(* Logix 5000 project; controller Comas_L4 vendor 1 type 14 code 193 rev 30.11; software revision 30.02; part 4 of 12 *)

ADD_ON_INSTRUCTION Output_Cams   (* revision 1.1, vendor Rockwell Automation *)
// Help:
// Cet Add-On permet la gestion d'une sortie commandée en fonction de la position d'un axe.
// Entre autre, la gestion des temps de réaction est prise en compte pour  le On/Off de la sortie.( Compensation du temps mort).
// La OutputCam est commandée quelque soit le sens de rotation de l'axe.( Bidirectionnal)
// Les entrées :
// In_ServoPosAxe_02.CommandPosition
VAR_INPUT
   Cmd_Enable_AOI : BOOL; {required}   // Entrée de Validation Du Fonctionnement De Output_Cam
   In_ServoPos : REAL; {required}   // Entrée de la Position de l'axe, préferez la Position Commandée
   In_ServoVel : REAL; {required}   // Entrée de la Vitesse de l'axe, Préferez la vitesse commandée
   Set_Period : REAL; {required}   // Entrée pour la Période de l'axe (Unwind Position) pour un axe rotatif. Pour un Axe Linéaire, Entrez ZERO comme valeur
   Set_OnPos : REAL; {required}   // Entrée pour la position de mise à UN de OuputCam
   Set_OffPos : REAL; {required}   // Entrée pour la position de mise à ZERO de OuputCam
   Set_TCompOn : DINT; {required}   // Entrée pour le temps de réaction de mise à UN des Actionneur/Pré-actionneur. ( en ms)
   Set_TCompOff : DINT; {required}   // Entrée pour le temps de réaction de mise à ZERO des Actionneur/Pré-actionneur.( en ms)
END_VAR
VAR_OUTPUT
   Out_Cam : BOOL; {access Read Only, required}   // Sotrie de la OutputCam
END_VAR
VAR
   L_OffPos : REAL;   // Pour Calcul de la position On avec Compensation du temps Mort
   L_OnPos : REAL;   // Pour Calcul de la position Off avec Compensation du temps Mort
END_VAR

ROUTINE Logic   (* structured text *)
   (*
   
   		Historic :
   
   					02.11.2008	PLM		Creation
   
   		Topic : This Add_On allows to switch On and Off anOutput and this related to the position of an Axis.
   				The deadTime compesation is taken into account ;
   *)
   
   
   
   	IF Cmd_Enable_AOI THEN
   
   		L_OnPos			:= Set_OnPos - (Set_TCompOn*In_ServoVel/1000);
   		IF L_OnPos < 0 THEN
   			L_OnPos			:= L_OnPos+Set_Period;
   		ELSIF L_OnPos > Set_Period THEN
   			L_OnPos			:= L_OnPos-Set_Period;
   		END_IF;
   
   
   		L_OffPos			:= Set_OffPos - (Set_TCompOff*In_ServoVel/1000);
   			IF L_OffPos < 0 THEN
   			L_OffPos		:= L_OffPos+Set_Period;
   		ELSIF L_OffPos > Set_Period THEN
   			L_OffPos		:= L_OffPos-Set_Period;
   		END_IF;
   
   		IF L_OnPos > L_OffPos THEN
   			IF In_ServoPos > L_OnPos OR In_ServoPos < L_OffPos THEN
   				Out_Cam		:= 1;
   			ELSE
   				Out_Cam		:= 0;
   			END_IF ;
   		ELSE
   			IF In_ServoPos > L_OnPos AND In_ServoPos < L_OffPos THEN
   				Out_Cam		:= 1;
   			ELSE
   				Out_Cam		:= 0;
   			END_IF ;
   		END_IF;
   	ELSE
   		Out_Cam				:= 0;
   	END_IF;
END_ROUTINE
END_ADD_ON_INSTRUCTION

ADD_ON_INSTRUCTION Pilotage_Relatif   (* revision 1.5 *)
// Revision note:
// V1.5: Guy : Mouvement incrémental
// V1.4: Guy : Simplification
// V1.3: Ajout:
//  tolérance, axe modulo
// V1.2: Avec mode de positionnement
// V1.1: Correction du double MSO
//    ( double appel de bloc)
// V1.0: Depart
VAR_IN_OUT
   MVT_Axe : AXIS_CIP_DRIVE; {required}   // Axe esclave a controler
END_VAR
VAR_INPUT
   MVT_Activation : BOOL; {required}   // Activation puissance A Activer avant d'engager
   MVT_Val_Position : REAL; {required}   // Position Cible
   MVT_Val_Vitesse : REAL; {required}   // Valeur de vitesse global de l'axe
   MVT_Val_Acc : REAL; {required}   // Valeur d accel gloable de laxe
   MVT_Val_Dec : REAL; {required}   // Valeur de decel
   MVT_Val_Jerk : REAL; {required}   // Valeur de jerk
END_VAR
VAR_OUTPUT
   MVT_ER : BOOL; {access Read Only, visible}   // Erreur dans le module
   MVT_En_Pos : BOOL; {visible}   // En position
END_VAR
VAR_INPUT
   MVT_Mode_Positionnement : DINT; {required}   // Mode de positionnement
   MVT_Tolerance_Arret : REAL; {required}   // tolerance d'arret
   MVT_Axe_Modulo : BOOL; {required}   // = 1 axe modulo
   MVT_Val_Modulo : DINT; {required}   // valeur du modulo
END_VAR
VAR_OUTPUT
   MVT_Axe_En_Mvt : BOOL; {access Read Only, visible}   // Axe en mouvement
END_VAR
VAR_INPUT
   MVT_Start : BOOL; {required}
END_VAR
VAR
   MVT_MSO_activation : MOTION_INSTRUCTION; {access None}
   MVT_Axe_Active : BOOL; {access None}
   MVT_MSO_desactivation : MOTION_INSTRUCTION; {access None}
   MVT_Val_Position_Neg : REAL; {access None}
   MVT_Val_Position_Pos : REAL; {access None}
   MVT_Commande_Mouvement : BOOL; {access None}
   MVT_MAM_Axe : MOTION_INSTRUCTION; {access None}
   MVT_MSO_desactivation2 : MOTION_INSTRUCTION; {access None}
   MVT_Val_Position_Neg_mod : REAL; {access None}
   MVT_Val_Position_Pos_mod : REAL; {access None}
   MVT_En_Pos_sans_modulo : BOOL; {access None}
   MVT_En_Pos_modulo : BOOL; {access None}
   MVT_Front_arret : BOOL; {access None}
   MVT_MAS_Axe : MOTION_INSTRUCTION; {access None}
   Front_Raz_Position : BOOL; {access None}
   MVT_Tempo_Axe_Actif : TIMER; {access None}
   MVT_Tempo_Axe_Actif_MSF : TIMER; {access None}
   Axe_En_Pos : BOOL; {access None}
   Etape_MAM : DINT; {access None}
   Frt_MAM_dn : BOOL; {access None}
   Frt_MAM_IP : BOOL; {access None}
   MVT_MAS : MOTION_INSTRUCTION; {access None}
END_VAR

ROUTINE Logic   (* ladder *)
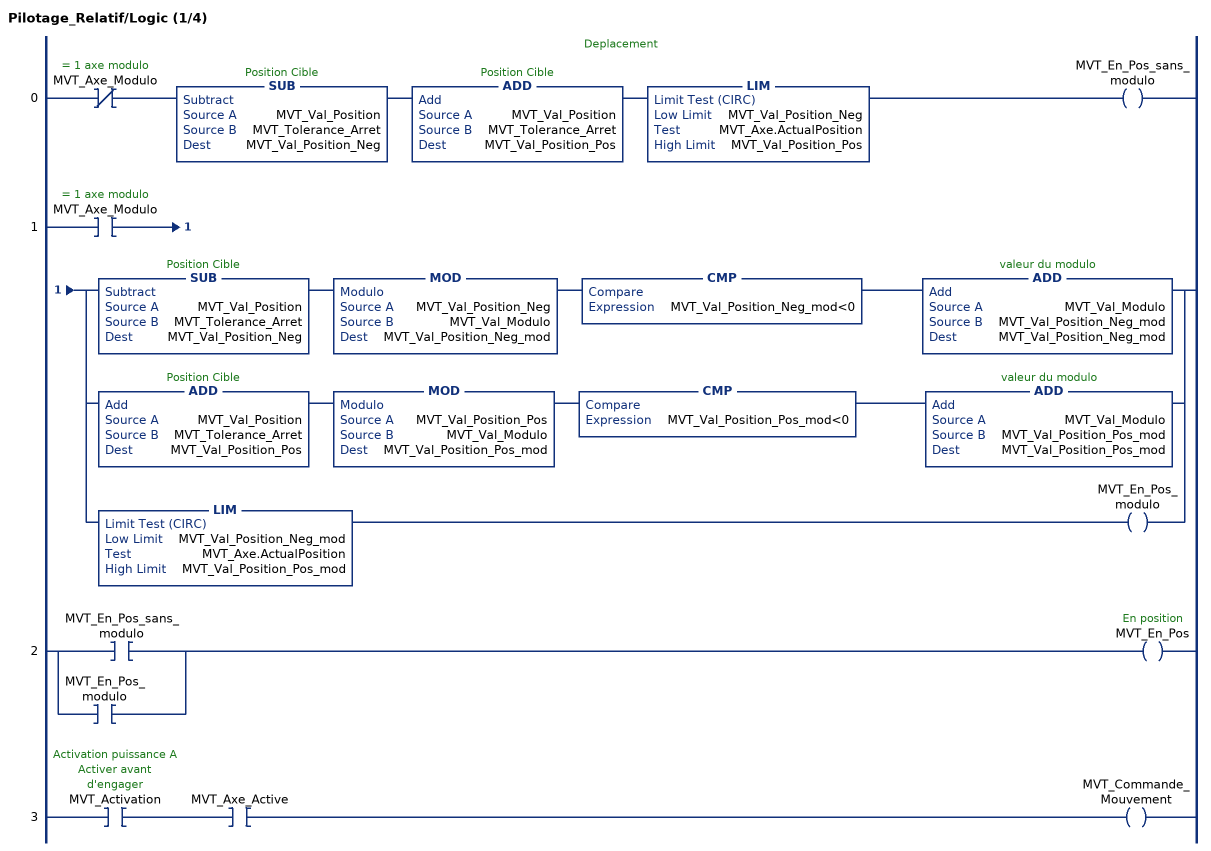
   // Deplacement
   0: XIO(MVT_Axe_Modulo)SUB(MVT_Val_Position,MVT_Tolerance_Arret,MVT_Val_Position_Neg)ADD(MVT_Val_Position,MVT_Tolerance_Arret,MVT_Val_Position_Pos)LIM(MVT_Val_Position_Neg,MVT_Axe.ActualPosition,MVT_Val_Position_Pos)OTE(MVT_En_Pos_sans_modulo);
   1: XIC(MVT_Axe_Modulo)[SUB(MVT_Val_Position,MVT_Tolerance_Arret,MVT_Val_Position_Neg) MOD(MVT_Val_Position_Neg,MVT_Val_Modulo,MVT_Val_Position_Neg_mod) CMP(MVT_Val_Position_Neg_mod<0) ADD(MVT_Val_Modulo,MVT_Val_Position_Neg_mod,MVT_Val_Position_Neg_mod) ,ADD(MVT_Val_Position,MVT_Tolerance_Arret,MVT_Val_Position_Pos) MOD(MVT_Val_Position_Pos,MVT_Val_Modulo,MVT_Val_Position_Pos_mod) CMP(MVT_Val_Position_Pos_mod<0) ADD(MVT_Val_Modulo,MVT_Val_Position_Pos_mod,MVT_Val_Position_Pos_mod) ,LIM(MVT_Val_Position_Neg_mod,MVT_Axe.ActualPosition,MVT_Val_Position_Pos_mod) OTE(MVT_En_Pos_modulo) ];
   2: [XIC(MVT_En_Pos_sans_modulo) ,XIC(MVT_En_Pos_modulo) ]OTE(MVT_En_Pos);
   3: XIC(MVT_Activation)XIC(MVT_Axe_Active)OTE(MVT_Commande_Mouvement);
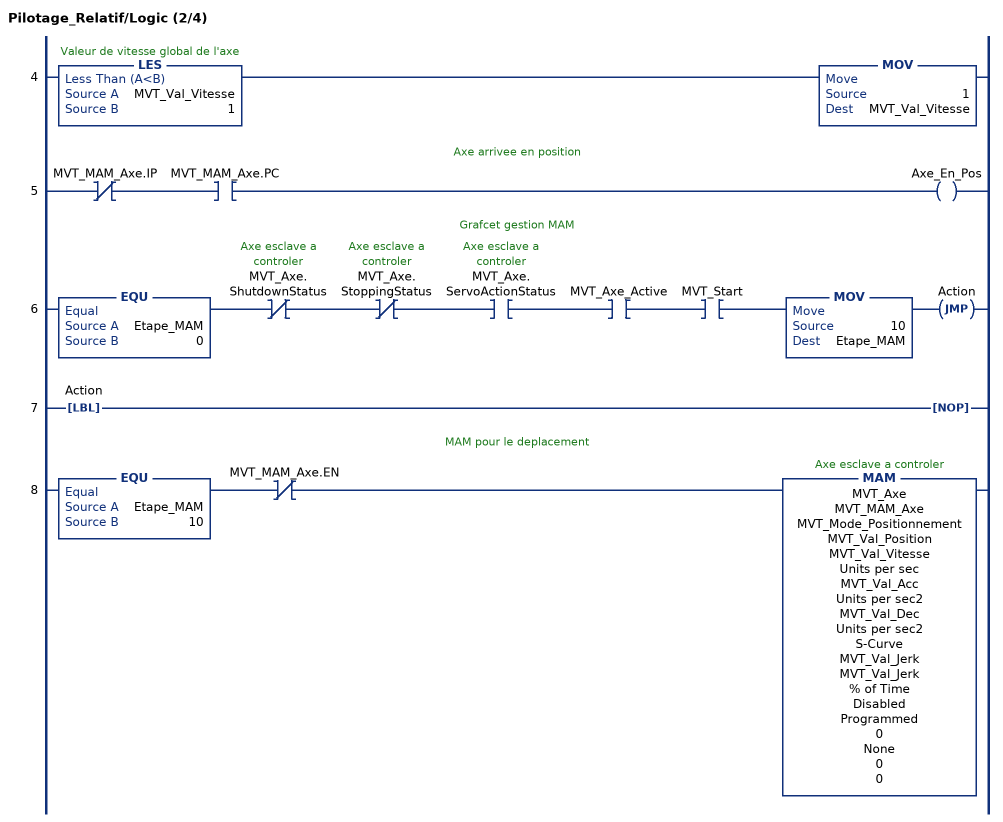
   4: LES(MVT_Val_Vitesse,1)MOV(1,MVT_Val_Vitesse);
   // Axe arrivee en position
   5: XIO(MVT_MAM_Axe.IP)XIC(MVT_MAM_Axe.PC)OTE(Axe_En_Pos);
   // Grafcet gestion MAM
   6: EQU(Etape_MAM,0)XIO(MVT_Axe.ShutdownStatus)XIO(MVT_Axe.StoppingStatus)XIC(MVT_Axe.ServoActionStatus)XIC(MVT_Axe_Active)XIC(MVT_Start)MOV(10,Etape_MAM)JMP(Action);
   7: LBL(Action)NOP();
   // MAM pour le deplacement
   8: EQU(Etape_MAM,10)XIO(MVT_MAM_Axe.EN)MAM(MVT_Axe,MVT_MAM_Axe,MVT_Mode_Positionnement,MVT_Val_Position,MVT_Val_Vitesse,Units per sec,MVT_Val_Acc,Units per sec2,MVT_Val_Dec,Units per sec2,S-Curve,MVT_Val_Jerk,MVT_Val_Jerk,% of Time,Disabled,Programmed,0,None,0,0);
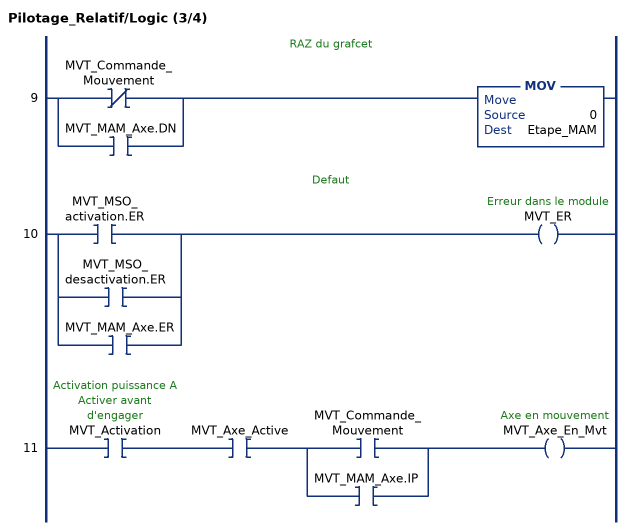
   // RAZ du grafcet
   9: [XIO(MVT_Commande_Mouvement) ,XIC(MVT_MAM_Axe.DN) ]MOV(0,Etape_MAM);
   // Defaut
   10: [XIC(MVT_MSO_activation.ER) ,XIC(MVT_MSO_desactivation.ER) ,XIC(MVT_MAM_Axe.ER) ]OTE(MVT_ER);
   11: XIC(MVT_Activation)XIC(MVT_Axe_Active)[XIC(MVT_Commande_Mouvement) ,XIC(MVT_MAM_Axe.IP) ]OTE(MVT_Axe_En_Mvt);
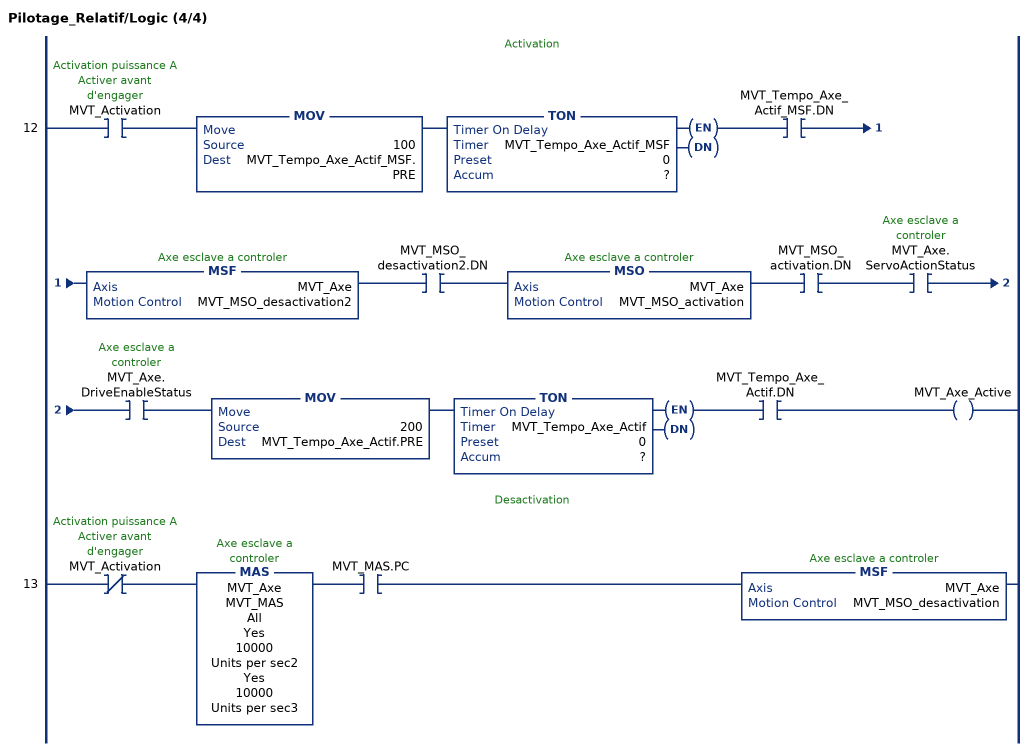
   // Activation
   12: XIC(MVT_Activation)MOV(100,MVT_Tempo_Axe_Actif_MSF.PRE)TON(MVT_Tempo_Axe_Actif_MSF,?,?)XIC(MVT_Tempo_Axe_Actif_MSF.DN)MSF(MVT_Axe,MVT_MSO_desactivation2)XIC(MVT_MSO_desactivation2.DN)MSO(MVT_Axe,MVT_MSO_activation)XIC(MVT_MSO_activation.DN)XIC(MVT_Axe.ServoActionStatus)XIC(MVT_Axe.DriveEnableStatus)MOV(200,MVT_Tempo_Axe_Actif.PRE)TON(MVT_Tempo_Axe_Actif,?,?)XIC(MVT_Tempo_Axe_Actif.DN)OTE(MVT_Axe_Active);
   // Desactivation
   13: XIO(MVT_Activation)MAS(MVT_Axe,MVT_MAS,All,Yes,10000,Units per sec2,Yes,10000,Units per sec3)XIC(MVT_MAS.PC)MSF(MVT_Axe,MVT_MSO_desactivation);
END_ROUTINE
END_ADD_ON_INSTRUCTION

ADD_ON_INSTRUCTION Pilotage_Relatif_Virtuel   (* revision 1.5 *)
// Revision note:
// V1.5: Guy : Mouvement incrémental
// V1.4: Guy : Simplification
// V1.3: Ajout:
//  tolérance, axe modulo
// V1.2: Avec mode de positionnement
// V1.1: Correction du double MSO
//    ( double appel de bloc)
// V1.0: Depart
VAR_IN_OUT
   MVT_Axe : AXIS_VIRTUAL; {required}   // Axe esclave a controler
END_VAR
VAR_INPUT
   MVT_Activation : BOOL; {required}   // Activation puissance A Activer avant d'engager
   MVT_Val_Position : REAL; {required}   // Position Cible
   MVT_Val_Vitesse : REAL; {required}   // Valeur de vitesse global de l'axe
   MVT_Val_Acc : REAL; {required}   // Valeur d accel gloable de laxe
   MVT_Val_Dec : REAL; {required}   // Valeur de decel
   MVT_Val_Jerk : REAL; {required}   // Valeur de jerk
END_VAR
VAR_OUTPUT
   MVT_ER : BOOL; {access Read Only, visible}   // Erreur dans le module
   MVT_En_Pos : BOOL; {visible}   // En position
END_VAR
VAR_INPUT
   MVT_Mode_Positionnement : DINT; {required}   // Mode de positionnement
   MVT_Tolerance_Arret : REAL; {required}   // tolerance d'arret
   MVT_Axe_Modulo : BOOL; {required}   // = 1 axe modulo
   MVT_Val_Modulo : DINT; {required}   // valeur du modulo
END_VAR
VAR_OUTPUT
   MVT_Axe_En_Mvt : BOOL; {access Read Only, visible}   // Axe en mouvement
END_VAR
VAR_INPUT
   MVT_Start : BOOL; {required}
END_VAR
VAR
   MVT_Axe_Active : BOOL; {access None}
   MVT_Val_Position_Neg : REAL; {access None}
   MVT_Val_Position_Pos : REAL; {access None}
   MVT_Commande_Mouvement : BOOL; {access None}
   MVT_MAM_Axe : MOTION_INSTRUCTION; {access None}
   MVT_Val_Position_Neg_mod : REAL; {access None}
   MVT_Val_Position_Pos_mod : REAL; {access None}
   MVT_En_Pos_sans_modulo : BOOL; {access None}
   MVT_En_Pos_modulo : BOOL; {access None}
   MVT_Front_arret : BOOL; {access None}
   MVT_MAS_Axe : MOTION_INSTRUCTION; {access None}
   Front_Raz_Position : BOOL; {access None}
   Axe_En_Pos : BOOL; {access None}
   Etape_MAM : DINT; {access None}
   Frt_MAM_dn : BOOL; {access None}
   Frt_MAM_IP : BOOL; {access None}
   MAS_1_AXE : MOTION_INSTRUCTION; {access None}
END_VAR

ROUTINE Logic   (* ladder *)
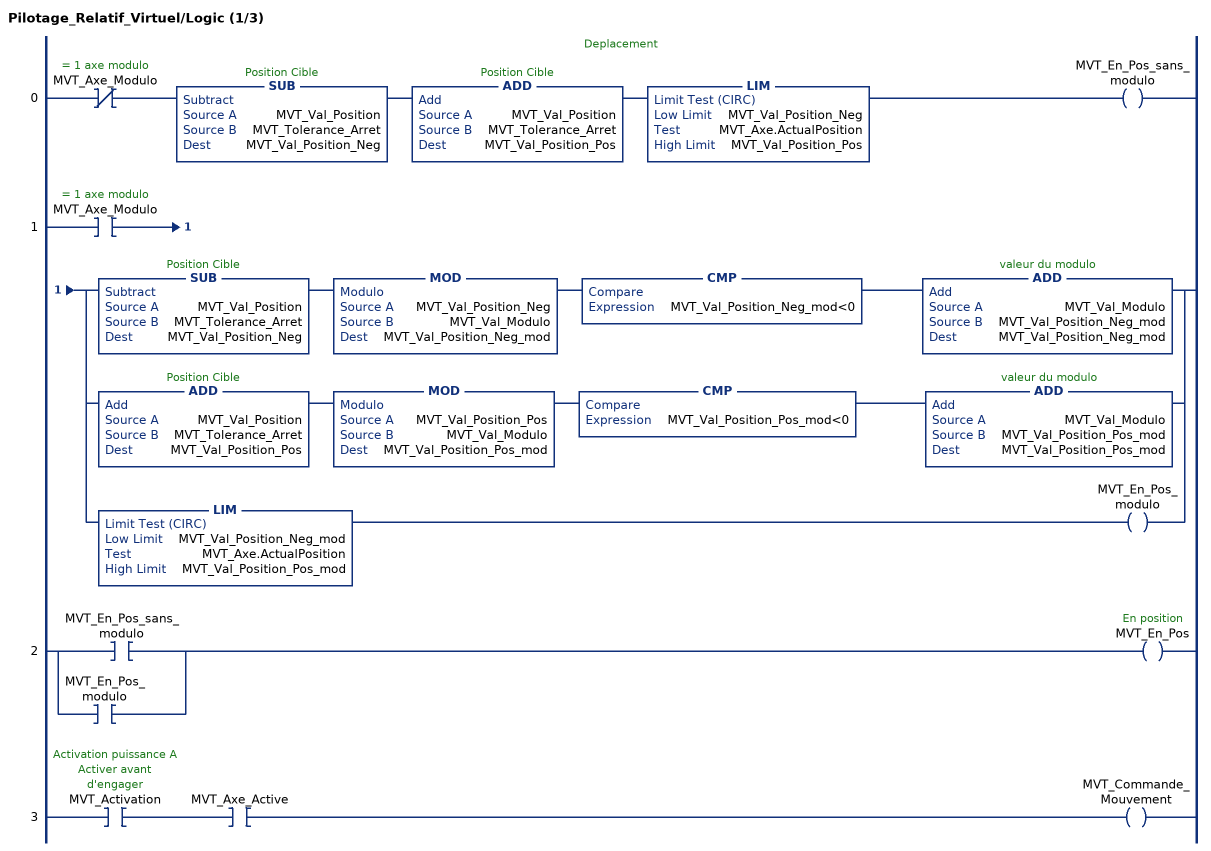
   // Deplacement
   0: XIO(MVT_Axe_Modulo)SUB(MVT_Val_Position,MVT_Tolerance_Arret,MVT_Val_Position_Neg)ADD(MVT_Val_Position,MVT_Tolerance_Arret,MVT_Val_Position_Pos)LIM(MVT_Val_Position_Neg,MVT_Axe.ActualPosition,MVT_Val_Position_Pos)OTE(MVT_En_Pos_sans_modulo);
   1: XIC(MVT_Axe_Modulo)[SUB(MVT_Val_Position,MVT_Tolerance_Arret,MVT_Val_Position_Neg) MOD(MVT_Val_Position_Neg,MVT_Val_Modulo,MVT_Val_Position_Neg_mod) CMP(MVT_Val_Position_Neg_mod<0) ADD(MVT_Val_Modulo,MVT_Val_Position_Neg_mod,MVT_Val_Position_Neg_mod) ,ADD(MVT_Val_Position,MVT_Tolerance_Arret,MVT_Val_Position_Pos) MOD(MVT_Val_Position_Pos,MVT_Val_Modulo,MVT_Val_Position_Pos_mod) CMP(MVT_Val_Position_Pos_mod<0) ADD(MVT_Val_Modulo,MVT_Val_Position_Pos_mod,MVT_Val_Position_Pos_mod) ,LIM(MVT_Val_Position_Neg_mod,MVT_Axe.ActualPosition,MVT_Val_Position_Pos_mod) OTE(MVT_En_Pos_modulo) ];
   2: [XIC(MVT_En_Pos_sans_modulo) ,XIC(MVT_En_Pos_modulo) ]OTE(MVT_En_Pos);
   3: XIC(MVT_Activation)XIC(MVT_Axe_Active)OTE(MVT_Commande_Mouvement);
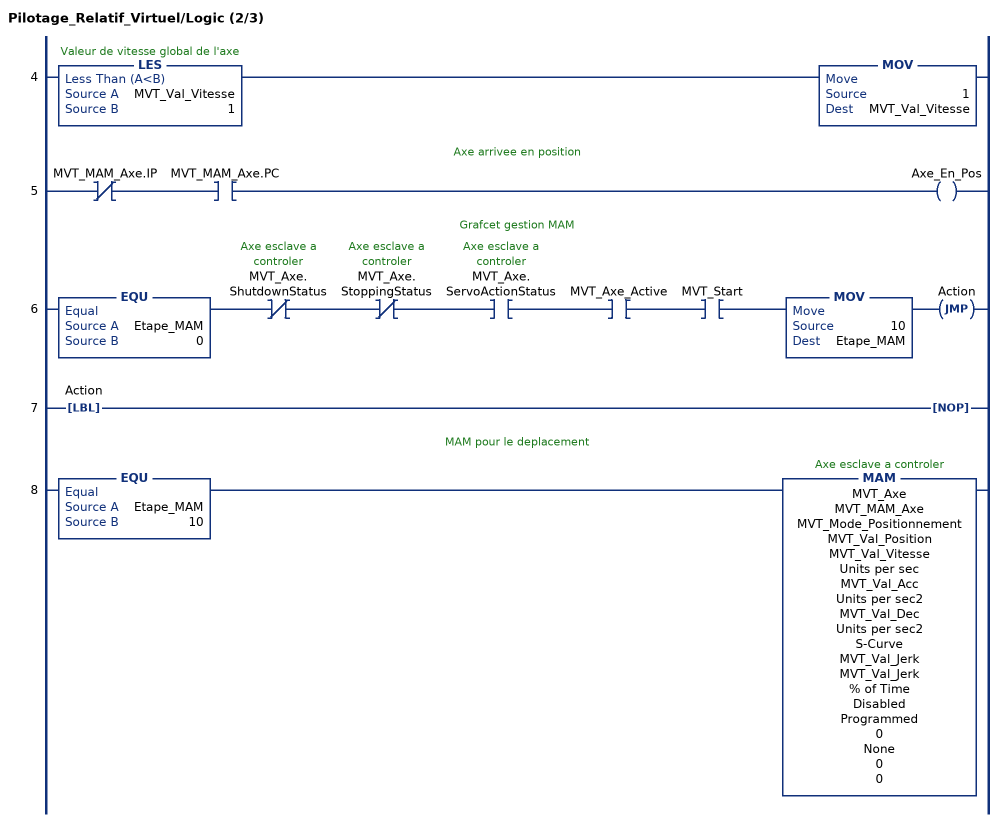
   4: LES(MVT_Val_Vitesse,1)MOV(1,MVT_Val_Vitesse);
   // Axe arrivee en position
   5: XIO(MVT_MAM_Axe.IP)XIC(MVT_MAM_Axe.PC)OTE(Axe_En_Pos);
   // Grafcet gestion MAM
   6: EQU(Etape_MAM,0)XIO(MVT_Axe.ShutdownStatus)XIO(MVT_Axe.StoppingStatus)XIC(MVT_Axe.ServoActionStatus)XIC(MVT_Axe_Active)XIC(MVT_Start)MOV(10,Etape_MAM)JMP(Action);
   7: LBL(Action)NOP();
   // MAM pour le deplacement
   8: EQU(Etape_MAM,10)MAM(MVT_Axe,MVT_MAM_Axe,MVT_Mode_Positionnement,MVT_Val_Position,MVT_Val_Vitesse,Units per sec,MVT_Val_Acc,Units per sec2,MVT_Val_Dec,Units per sec2,S-Curve,MVT_Val_Jerk,MVT_Val_Jerk,% of Time,Disabled,Programmed,0,None,0,0);
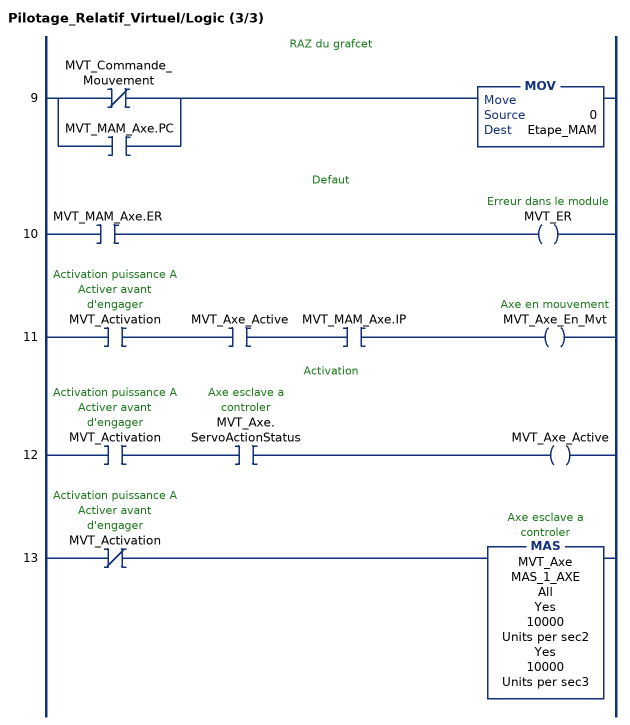
   // RAZ du grafcet
   9: [XIO(MVT_Commande_Mouvement) ,XIC(MVT_MAM_Axe.PC) ]MOV(0,Etape_MAM);
   // Defaut
   10: XIC(MVT_MAM_Axe.ER)OTE(MVT_ER);
   11: XIC(MVT_Activation)XIC(MVT_Axe_Active)XIC(MVT_MAM_Axe.IP)OTE(MVT_Axe_En_Mvt);
   // Activation
   12: XIC(MVT_Activation)XIC(MVT_Axe.ServoActionStatus)OTE(MVT_Axe_Active);
   13: XIO(MVT_Activation)MAS(MVT_Axe,MAS_1_AXE,All,Yes,10000,Units per sec2,Yes,10000,Units per sec3);
END_ROUTINE
END_ADD_ON_INSTRUCTION

ADD_ON_INSTRUCTION Pilotage_Vitesse_Rapide_V4   (* revision 1.4 *)
// Revision note:
// V1: Version initiale :
// V1-2:
// - Correction MASR / MAFR
// - Correction gestion Graphcet
// V1-4: ROD
// - Optimisation vitesse de scan
VAR_IN_OUT
   Axe : AXIS_VIRTUAL; {required}
END_VAR
VAR_INPUT
   Vitesse : REAL; {visible}
   Acc : REAL; {visible}
   Dec : REAL; {visible}
   Jerk : REAL; {visible}
   Autorisation : BOOL; {visible}
   Acquit : BOOL; {visible}
   Defaut_axe : BOOL; {visible}
END_VAR
VAR_OUTPUT
   St_Erreur : BOOL; {visible}
   St_En_Attente : BOOL; {visible}
   St_Init1 : BOOL; {visible}
   St_Init2 : BOOL; {visible}
   St_Activation : BOOL; {visible}
   St_Vitesse : BOOL; {visible}
   St_Arret : BOOL; {visible}
   St_Desactivation : BOOL; {visible}
END_VAR
VAR
   Graph : DINT; {access None}
   Axe_Actif : BOOL; {access None}
   Motion_Control_MAJ : MOTION_INSTRUCTION; {access None}
   Motion_Control_MAFR : MOTION_INSTRUCTION; {access None}
   Motion_Control_MASR : MOTION_INSTRUCTION; {access None}
   Motion_Control_MSO : MOTION_INSTRUCTION; {access None}
   Motion_Control_MAS1 : MOTION_INSTRUCTION; {access None}
   Motion_Control_MAS2 : MOTION_INSTRUCTION; {access None}
   Motion_Control_MSF1 : MOTION_INSTRUCTION; {access None}
   Motion_Control_MSF2 : MOTION_INSTRUCTION; {access None}
   Motion_Control_MAS3 : MOTION_INSTRUCTION; {access None}
   Memo_Graph_20 : BOOL; {access None}
   Memo_Graph_60 : BOOL; {access None}
   Timeout_Graph : FBD_TIMER; {access None}
   Erreur_Timeout_Controle : BOOL; {access None}
   Front_Acquit_Defaut : FBD_ONESHOT; {access None}
END_VAR

ROUTINE Logic   (* structured text *)
   // ////////////////////////////////////////////////////////
   // Defaut
   // ////////////////////////////////////////////////////////
   IF	(Motion_Control_MASR.ER OR Motion_Control_MAFR.ER OR Motion_Control_MAS1.ER OR Motion_Control_MSO.ER) OR
   		(Motion_Control_MAJ.ER OR Motion_Control_MAS2.ER OR Motion_Control_MSF1.ER OR Defaut_axe) AND NOT St_Erreur THEN
   		Motion_Control_MASR.FLAGS	:= 0;
   		Motion_Control_MAFR.FLAGS	:= 0;
   		Motion_Control_MAS1.FLAGS	:= 0;
   		Motion_Control_MSO.FLAGS	:= 0;
   		Motion_Control_MAJ.FLAGS	:= 0;
   		Motion_Control_MAS2.FLAGS	:= 0;
   		Motion_Control_MSF1.FLAGS	:= 0;
   		Graph:=0;
   		St_Erreur:=1;
   		MAS(Axe,
   			Motion_Control_MAS3,
   			All,
   			Yes,
   			Dec ,
   			Unitspersec2,
   			Yes,
   			Jerk,
   			%ofTime);
   END_IF;
   
   // Acquit Defaut
   IF Acquit OR Front_Acquit_Defaut.OutputBit THEN
   	St_Erreur:=0;
   END_IF;
   
   Front_Acquit_Defaut.InputBit :=Autorisation;
   OSRI(Front_Acquit_Defaut);
   
   
   // ////////////////////////////////////////////////////////
   // Etat
   // ////////////////////////////////////////////////////////
   St_En_Attente:=0;
   St_Init1:=0;
   St_Init2:=0;
   St_Activation:=0;
   St_Vitesse:=0;
   St_Arret:=0;
   St_Desactivation:=0;
   
   // ////////////////////////////////////////////////////////
   // Cycle
   // ////////////////////////////////////////////////////////
   CASE Graph OF
   	// Depart
   	0:
   		St_En_Attente:=1;
   		IF Autorisation AND NOT Axe.StoppingStatus AND NOT Defaut_axe AND NOT St_Erreur THEN
   			Graph:=5;
   		END_IF;
   
   	// Init des etats
   	3:
   		St_Init1:=1;
   		// Init des etats
   		Motion_Control_MASR.FLAGS	:= 0;
   		Motion_Control_MAFR.FLAGS	:= 0;
   		Motion_Control_MAS1.FLAGS	:= 0;
   		Motion_Control_MSO.FLAGS	:= 0;
   		Motion_Control_MAJ.FLAGS	:= 0;
   		Motion_Control_MAS2.FLAGS	:= 0;
   		Motion_Control_MSF1.FLAGS	:= 0;
   		// Acquit des erreurs
   		St_Erreur:=0;
   
   	// Motion Reset Shutdown status
   	5:
   		St_Init1:=1;
   		Graph:=7;
   
   	// Motion Clear Fault
   	7:
   		St_Init1:=1;
   		Graph:=10;
   
   	// Arret si mouvement en cours
   	10:
   		St_Init2:=1;
   		IF NOT Motion_Control_MAS1.EN THEN
   			MAS(Axe,
   					Motion_Control_MAS1,
   					All,
   					Yes,
   					Dec ,
   					Unitspersec2,
   					Yes,
   					Jerk,
   					%ofTime);
   		END_IF;
   		// Condition
   		IF Motion_Control_MAS1.EN AND Motion_Control_MAS1.DN AND NOT Motion_Control_MAS1.IP AND NOT Axe.StoppingStatus THEN
   			Graph:=30;
   		END_IF;
   
   	// Activation
   	20:
   
   	// Activation
   	25:
   
   	// Vitesse
   	30:
   		St_Vitesse:=1;
   		MAJ(Axe,
   		Motion_Control_MAJ,
   		0,
   		Vitesse,
   		0,
   		Acc,
   		0,
   		Dec,
   		0,
   		0,
   		Jerk,
   		Jerk,
   		%ofTime,
   		0,			// Modifie pour controle via mam
   		0,0,None);
   		// Conditions
   		Graph:=40;
   
   	// Arret ou vitesse
   	40:
   		St_Vitesse:=1;
   		IF NOT Autorisation THEN
   			Graph:=50;
   		ELSE
   			Graph:=30;
   		END_IF;
   
   	// Arret
   	50:
   		St_Arret:=1;
   		IF NOT Motion_Control_MAS2.EN THEN
   			MAS(Axe,
   			Motion_Control_MAS2,
   			All,
   			Yes,
   			Dec ,
   			Unitspersec2,
   			Yes,
   			Jerk,
   			%ofTime);
   		END_IF;
   		// Condition
   		IF Motion_Control_MAS2.EN AND Motion_Control_MAS2.DN AND NOT Motion_Control_MAS2.IP AND NOT Axe.StoppingStatus THEN
   			Graph:=60;
   		END_IF;
   
   
   	// Desactivation
   	60:
   		St_Desactivation:=1;
   		Graph:=65;
   
   	// Desactivation
   	65:
   		St_Desactivation:=1;
   		// Init des etats
   		Motion_Control_MASR.FLAGS	:= 0;
   		Motion_Control_MAFR.FLAGS	:= 0;
   		Motion_Control_MAS1.FLAGS	:= 0;
   		Motion_Control_MSO.FLAGS	:= 0;
   		Motion_Control_MAJ.FLAGS	:= 0;
   		Motion_Control_MAS2.FLAGS	:= 0;
   		Motion_Control_MSF1.FLAGS	:= 0;
   		Graph:=0;
   END_CASE;
   
   // Mise a jour etat
   IF St_Erreur THEN
   	St_En_Attente:=0;
   END_If;
END_ROUTINE
END_ADD_ON_INSTRUCTION

ADD_ON_INSTRUCTION Raz_Axe   (* revision 1.2 *)
VAR_IN_OUT
   AXE : AXIS_CIP_DRIVE; {required}
END_VAR
VAR_INPUT
   RAZ : BOOL; {required}
   acc : REAL; {required}
   dec : REAL; {required}
   jerk : REAL; {required}
END_VAR
VAR_OUTPUT
   ER : BOOL; {access Read Only, visible}
END_VAR
VAR
   MASR_AXE : MOTION_INSTRUCTION;
   MAFR_AXE : MOTION_INSTRUCTION;
   MAS_AXE : MOTION_INSTRUCTION;
END_VAR

ROUTINE Logic   (* ladder *)
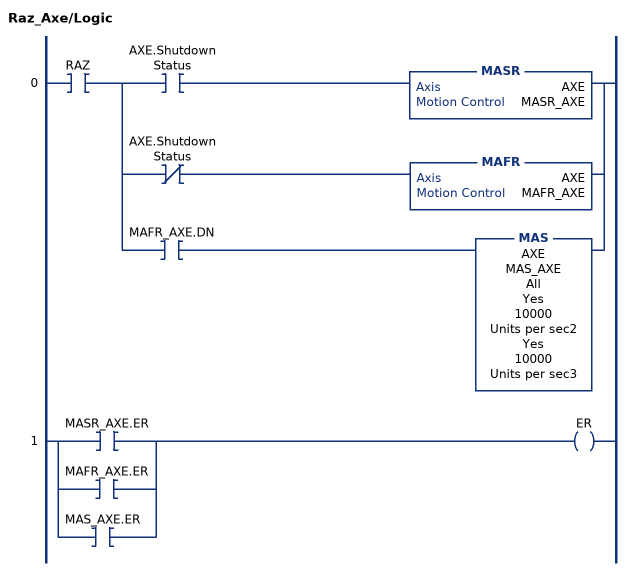
   0: XIC(RAZ)[XIC(AXE.ShutdownStatus) MASR(AXE,MASR_AXE) ,XIO(AXE.ShutdownStatus) MAFR(AXE,MAFR_AXE) ,XIC(MAFR_AXE.DN) MAS(AXE,MAS_AXE,All,Yes,10000,Units per sec2,Yes,10000,Units per sec3) ];
   1: [XIC(MASR_AXE.ER) ,XIC(MAFR_AXE.ER) ,XIC(MAS_AXE.ER) ]OTE(ER);
END_ROUTINE
END_ADD_ON_INSTRUCTION

ADD_ON_INSTRUCTION Registre_Avance_Convoyeur   (* revision 1.0 *)
// Distance_totale en m
// Anticipation en nombre de registre
// Coeff_avance [0:1000]
VAR_INPUT
   Presence_biscuit_E : BOOL;
END_VAR
VAR_OUTPUT
   Presence_biscuit_S : BOOL;
END_VAR
VAR_INPUT
   Distance_totale : DINT; {required}
   Anticipation_arret : INT; {required}
END_VAR
VAR_OUTPUT
   Erreur_anticipation_arret : BOOL; {access None, visible}
   Erreur_anticipation_marche : BOOL; {access None, visible}
END_VAR
VAR_INPUT
   Anticipation_marche : INT; {access None, required}
   Coeff_avance : DINT; {access None, required}
END_VAR
VAR_OUTPUT
   Marche : BOOL; {access None, visible}
END_VAR
VAR_INPUT
   Coeff_conv_Hz_mm : REAL; {required}
   Retour_Variateur : INT; {access None}
END_VAR
VAR
   Compteur : TIMER; {access None}
   Registre_100 : INT[128] := ([0] := 99); {access None}
   Registre_tmp : INT[128]; {access None}
   Distance_anticipation_arret : INT; {access None}
   Distance_anticipation_marche : INT; {access None}
   Compteur_Sortie : TIMER; {access None}
   Coeff_pas_registre : REAL; {access None}
   Distance_totale_registre : DINT; {access None}
   Frequence_moteur : DINT;
END_VAR

ROUTINE Logic   (* ladder *)
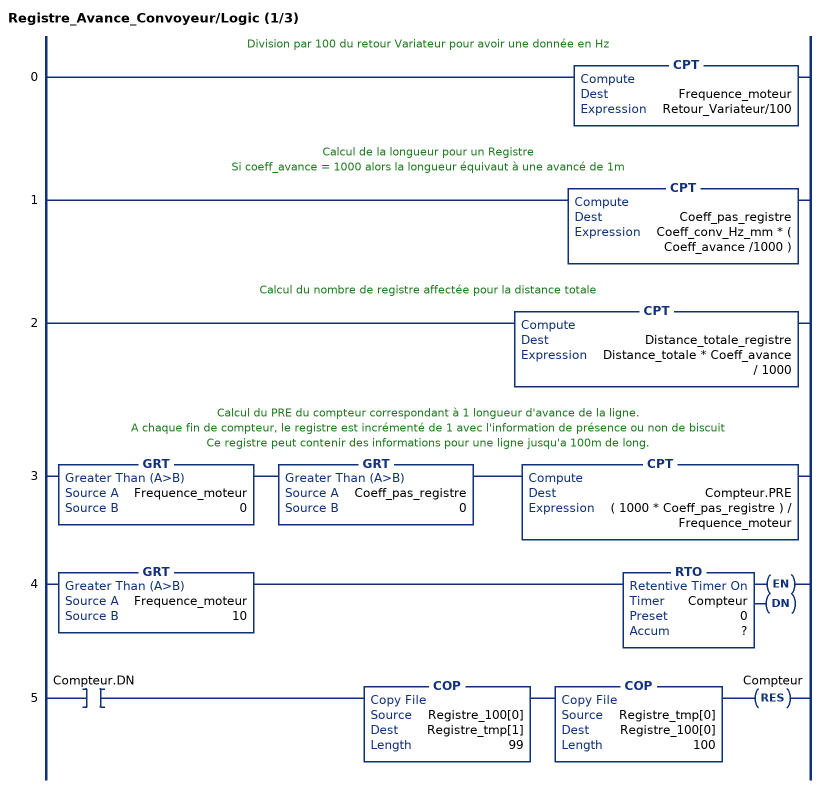
   // Division par 100 du retour Variateur pour avoir une donnée en Hz
   0: CPT(Frequence_moteur,Retour_Variateur/100);
   // Calcul de la longueur pour un Registre
   // Si coeff_avance = 1000 alors la longueur équivaut à une avancé de 1m
   1: CPT(Coeff_pas_registre,Coeff_conv_Hz_mm * ( Coeff_avance /1000 ));
   // Calcul du nombre de registre affectée pour la distance totale
   2: CPT(Distance_totale_registre,Distance_totale * Coeff_avance / 1000);
   // Calcul du PRE du compteur correspondant à 1 longueur d'avance de la ligne.
   // A chaque fin de compteur, le registre est incrémenté de 1 avec l'information de présence ou non de biscuit
   // Ce registre peut contenir des informations pour une ligne jusqu'a 100m de long.
   3: GRT(Frequence_moteur,0)GRT(Coeff_pas_registre,0)CPT(Compteur.PRE,( 1000 * Coeff_pas_registre ) / Frequence_moteur);
   4: GRT(Frequence_moteur,10)RTO(Compteur,?,?);
   5: XIC(Compteur.DN)COP(Registre_100[0],Registre_tmp[1],99)COP(Registre_tmp[0],Registre_100[0],100)RES(Compteur);
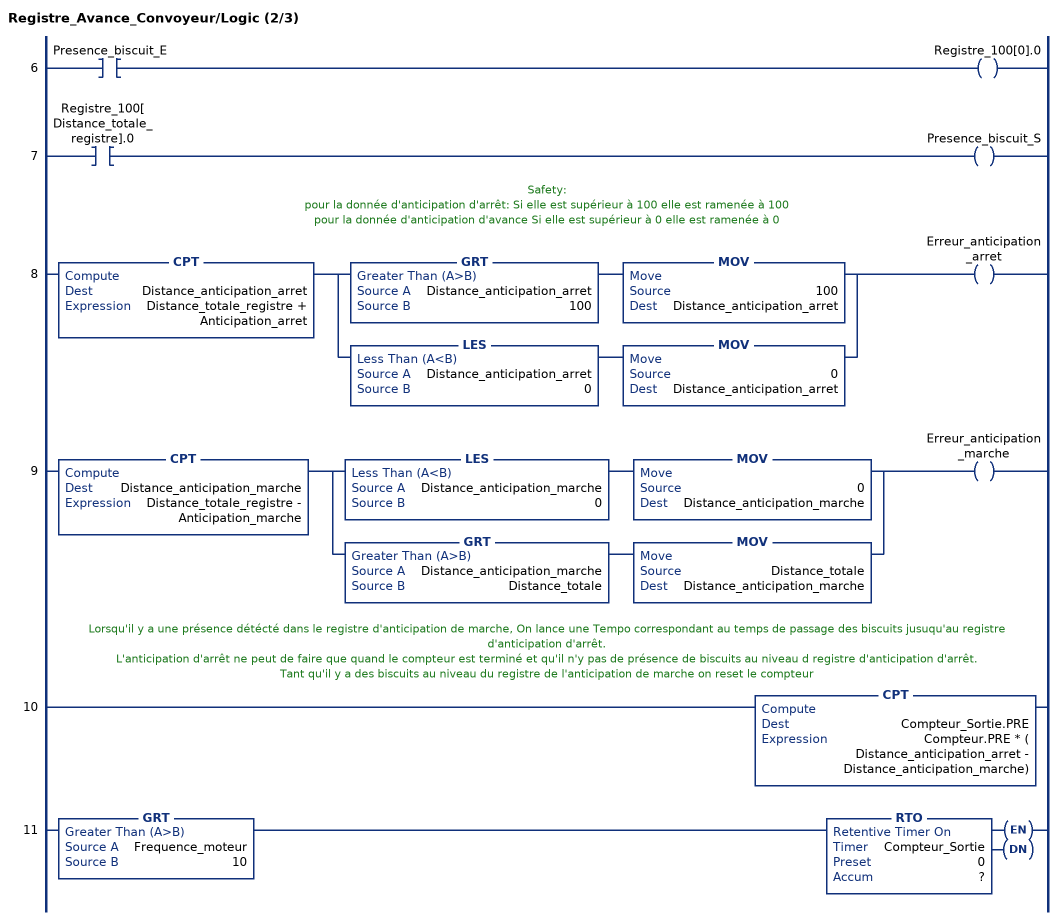
   6: XIC(Presence_biscuit_E)OTE(Registre_100[0].0);
   7: XIC(Registre_100[Distance_totale_registre].0)OTE(Presence_biscuit_S);
   // Safety:
   // pour la donnée d'anticipation d'arrêt: Si elle est supérieur à 100 elle est ramenée à 100
   // pour la donnée d'anticipation d'avance Si elle est supérieur à 0 elle est ramenée à 0
   8: CPT(Distance_anticipation_arret,Distance_totale_registre + Anticipation_arret)[GRT(Distance_anticipation_arret,100) MOV(100,Distance_anticipation_arret) ,LES(Distance_anticipation_arret,0) MOV(0,Distance_anticipation_arret) ]OTE(Erreur_anticipation_arret);
   9: CPT(Distance_anticipation_marche,Distance_totale_registre - Anticipation_marche)[LES(Distance_anticipation_marche,0) MOV(0,Distance_anticipation_marche) ,GRT(Distance_anticipation_marche,Distance_totale) MOV(Distance_totale,Distance_anticipation_marche) ]OTE(Erreur_anticipation_marche);
   // Lorsqu'il y a une présence détécté dans le registre d'anticipation de marche, On lance une Tempo correspondant au temps de passage des biscuits jusuqu'au registre d'anticipation d'arrêt.
   // L'anticipation d'arrêt ne peut de faire que quand le compteur est terminé et qu'il n'y pas de présence de biscuits au niveau d registre d'anticipation d'arrêt.
   // Tant qu'il y a des biscuits au niveau du registre de l'anticipation de marche on reset le compteur
   10: CPT(Compteur_Sortie.PRE,Compteur.PRE * ( Distance_anticipation_arret - Distance_anticipation_marche));
   11: GRT(Frequence_moteur,10)RTO(Compteur_Sortie,?,?);
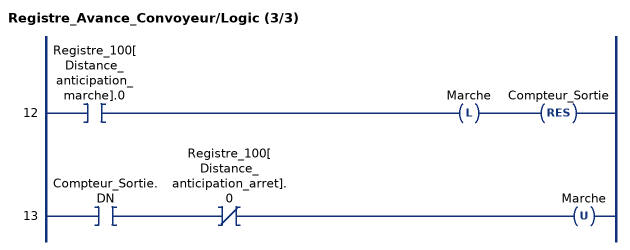
   12: XIC(Registre_100[Distance_anticipation_marche].0)OTL(Marche)RES(Compteur_Sortie);
   13: XIC(Compteur_Sortie.DN)XIO(Registre_100[Distance_anticipation_arret].0)OTU(Marche);
END_ROUTINE
END_ADD_ON_INSTRUCTION

ADD_ON_INSTRUCTION Registre_Avance_Convoyeur_V2   (* revision 1.0 *)
// Distance_totale en m
// Anticipation en nombre de registre
// Coeff_avance [0:1000]
VAR_INPUT
   Presence_biscuit_E : BOOL;
END_VAR
VAR_OUTPUT
   Presence_biscuit_S : BOOL;
END_VAR
VAR_INPUT
   Distance_totale : DINT; {required}
   Anticipation_arret : INT; {required}
END_VAR
VAR_OUTPUT
   Erreur_anticipation_arret : BOOL; {access None, visible}
   Erreur_anticipation_marche : BOOL; {access None, visible}
END_VAR
VAR_INPUT
   Anticipation_marche : INT; {access None, required}
   Coeff_avance : DINT; {access None, required}
END_VAR
VAR_OUTPUT
   Marche : BOOL; {access None, visible}
END_VAR
VAR_INPUT
   Coeff_conv_Hz_mm : REAL; {required}
   Retour_Variateur : INT; {access None}
END_VAR
VAR
   Compteur : TIMER; {access None}
   Registre_100 : INT[128] := ([0] := 99); {access None}
   Registre_tmp : INT[128]; {access None}
   Distance_anticipation_arret : INT; {access None}
   Distance_anticipation_marche : INT; {access None}
   Compteur_Sortie : TIMER; {access None}
   Coeff_pas_registre : REAL; {access None}
   Distance_totale_registre : DINT; {access None}
   Frequence_moteur : REAL;
END_VAR

ROUTINE Logic   (* ladder *)
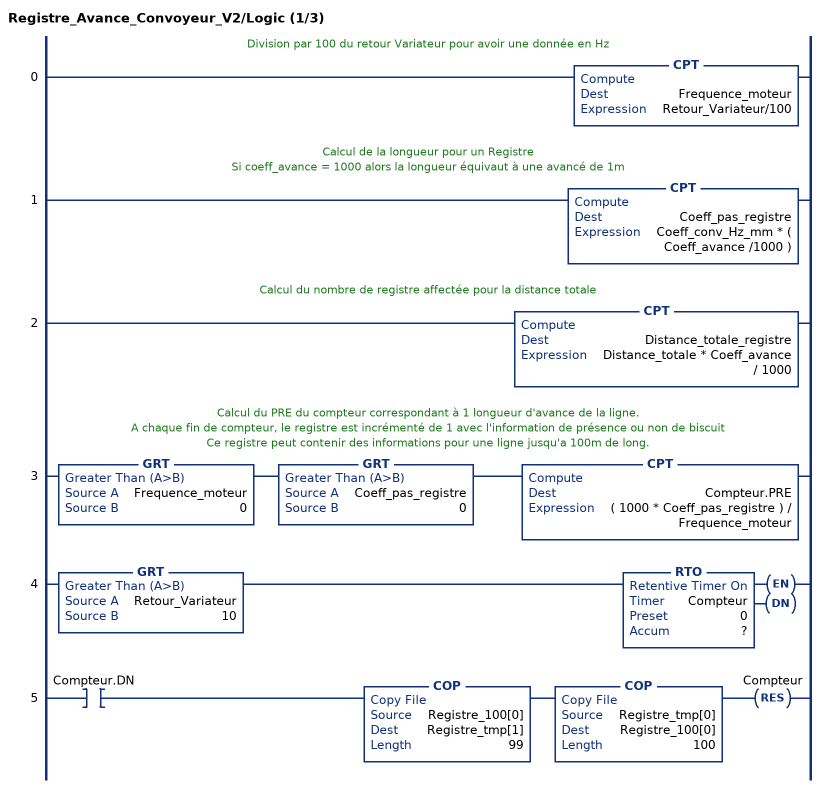
   // Division par 100 du retour Variateur pour avoir une donnée en Hz
   0: CPT(Frequence_moteur,Retour_Variateur/100);
   // Calcul de la longueur pour un Registre
   // Si coeff_avance = 1000 alors la longueur équivaut à une avancé de 1m
   1: CPT(Coeff_pas_registre,Coeff_conv_Hz_mm * ( Coeff_avance /1000 ));
   // Calcul du nombre de registre affectée pour la distance totale
   2: CPT(Distance_totale_registre,Distance_totale * Coeff_avance / 1000);
   // Calcul du PRE du compteur correspondant à 1 longueur d'avance de la ligne.
   // A chaque fin de compteur, le registre est incrémenté de 1 avec l'information de présence ou non de biscuit
   // Ce registre peut contenir des informations pour une ligne jusqu'a 100m de long.
   3: GRT(Frequence_moteur,0)GRT(Coeff_pas_registre,0)CPT(Compteur.PRE,( 1000 * Coeff_pas_registre ) / Frequence_moteur);
   4: GRT(Retour_Variateur,10)RTO(Compteur,?,?);
   5: XIC(Compteur.DN)COP(Registre_100[0],Registre_tmp[1],99)COP(Registre_tmp[0],Registre_100[0],100)RES(Compteur);
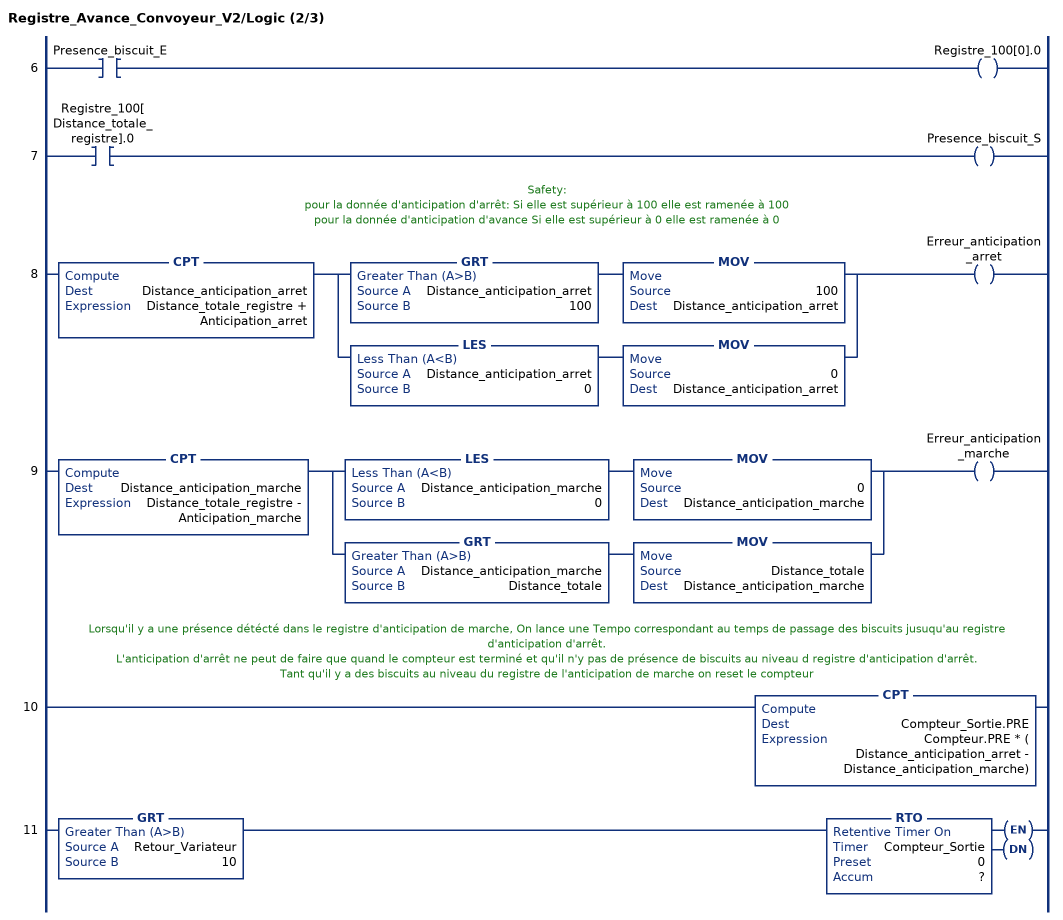
   6: XIC(Presence_biscuit_E)OTE(Registre_100[0].0);
   7: XIC(Registre_100[Distance_totale_registre].0)OTE(Presence_biscuit_S);
   // Safety:
   // pour la donnée d'anticipation d'arrêt: Si elle est supérieur à 100 elle est ramenée à 100
   // pour la donnée d'anticipation d'avance Si elle est supérieur à 0 elle est ramenée à 0
   8: CPT(Distance_anticipation_arret,Distance_totale_registre + Anticipation_arret)[GRT(Distance_anticipation_arret,100) MOV(100,Distance_anticipation_arret) ,LES(Distance_anticipation_arret,0) MOV(0,Distance_anticipation_arret) ]OTE(Erreur_anticipation_arret);
   9: CPT(Distance_anticipation_marche,Distance_totale_registre - Anticipation_marche)[LES(Distance_anticipation_marche,0) MOV(0,Distance_anticipation_marche) ,GRT(Distance_anticipation_marche,Distance_totale) MOV(Distance_totale,Distance_anticipation_marche) ]OTE(Erreur_anticipation_marche);
   // Lorsqu'il y a une présence détécté dans le registre d'anticipation de marche, On lance une Tempo correspondant au temps de passage des biscuits jusuqu'au registre d'anticipation d'arrêt.
   // L'anticipation d'arrêt ne peut de faire que quand le compteur est terminé et qu'il n'y pas de présence de biscuits au niveau d registre d'anticipation d'arrêt.
   // Tant qu'il y a des biscuits au niveau du registre de l'anticipation de marche on reset le compteur
   10: CPT(Compteur_Sortie.PRE,Compteur.PRE * ( Distance_anticipation_arret - Distance_anticipation_marche));
   11: GRT(Retour_Variateur,10)RTO(Compteur_Sortie,?,?);
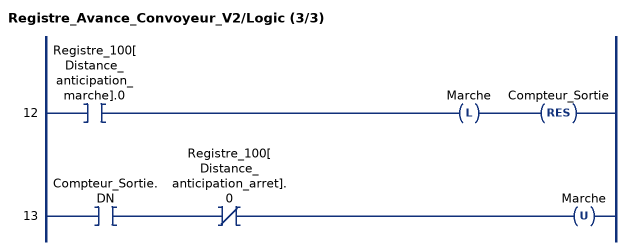
   12: XIC(Registre_100[Distance_anticipation_marche].0)OTL(Marche)RES(Compteur_Sortie);
   13: XIC(Compteur_Sortie.DN)XIO(Registre_100[Distance_anticipation_arret].0)OTU(Marche);
END_ROUTINE
END_ADD_ON_INSTRUCTION

ADD_ON_INSTRUCTION Test_Axe_Avec_Autorisation   (* revision 1.4 *)
// Revision note:
// V1.4 + Autorisation séparée
// V1.4: Correction MAS avec ACC/DEC
// V1.3: Suppression autorisation en entrée du bloc
// V1.2: Ajout init absolu
VAR_IN_OUT
   Axe : AXIS_CIP_DRIVE; {required}
END_VAR
VAR_INPUT
   Test_Positif : BOOL; {required}
   Test_Negatif : BOOL; {required}
   Vitesse : REAL; {required}
   Acc : REAL; {required}
   Dec : REAL; {required}
   Jerk : REAL; {required}
   Activation_Init : BOOL; {required}
   Etat_Init : BOOL; {required}
END_VAR
VAR_OUTPUT
   IP : BOOL; {access Read Only, visible}
   ER : BOOL; {access Read Only, visible}
   Init_OK : BOOL; {access Read Only, visible}
END_VAR
VAR_INPUT
   Autorisation : BOOL; {required}
END_VAR
VAR
   MAJ_Test : MOTION_INSTRUCTION;
   MSO_Test : MOTION_INSTRUCTION;
   Temp : BOOL;
   MSF_Test : MOTION_INSTRUCTION;
   MSO_Test_Positif : MOTION_INSTRUCTION;
   MSO_Test_negatif : MOTION_INSTRUCTION;
   MAJ_Test_Positif : MOTION_INSTRUCTION;
   MAJ_Test_Negatif : MOTION_INSTRUCTION;
   MASR_AXE : MOTION_INSTRUCTION;
   MAFR_AXE : MOTION_INSTRUCTION;
   MAS_AXE : MOTION_INSTRUCTION;
   TON_Test : TIMER;
   MCD_Jog : MOTION_INSTRUCTION;
   erreur_1 : BOOL;
   erreur_2 : BOOL;
   MAH_Axe : MOTION_INSTRUCTION;
   Vitesse_Sens : REAL;
   MAS2_AXE : MOTION_INSTRUCTION;
   temp2 : BOOL;
   TEMP10 : BOOL;
   MASMAH2_AXE : MOTION_INSTRUCTION;
   FRONTCPT : BOOL;
   INITENCOURS : BOOL;
   MSF_Test_INIT : MOTION_INSTRUCTION;
   MSO_Test_INIT : MOTION_INSTRUCTION;
   FRONTCPT2 : BOOL;
   Temp3 : BOOL;
   Temp4 : BOOL;
   Autor_MAJ : BOOL; {access None}
END_VAR

ROUTINE Logic   (* ladder *)
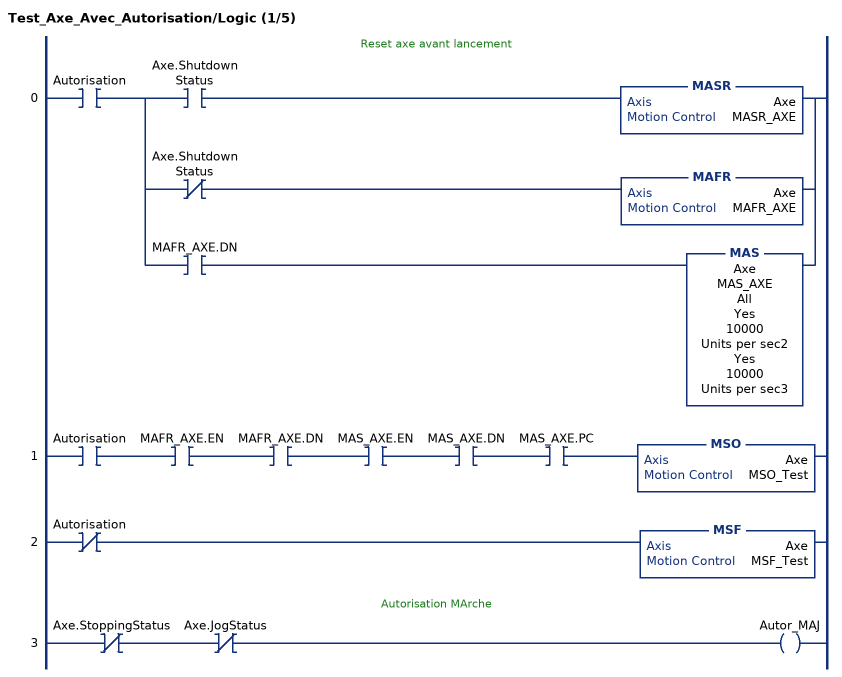
   // Reset axe avant lancement
   0: XIC(Autorisation)[XIC(Axe.ShutdownStatus) MASR(Axe,MASR_AXE) ,XIO(Axe.ShutdownStatus) MAFR(Axe,MAFR_AXE) ,XIC(MAFR_AXE.DN) MAS(Axe,MAS_AXE,All,Yes,10000,Units per sec2,Yes,10000,Units per sec3) ];
   1: XIC(Autorisation)XIC(MAFR_AXE.EN)XIC(MAFR_AXE.DN)XIC(MAS_AXE.EN)XIC(MAS_AXE.DN)XIC(MAS_AXE.PC)MSO(Axe,MSO_Test);
   2: XIO(Autorisation)MSF(Axe,MSF_Test);
   // Autorisation MArche
   3: XIO(Axe.StoppingStatus)XIO(Axe.JogStatus)OTE(Autor_MAJ);
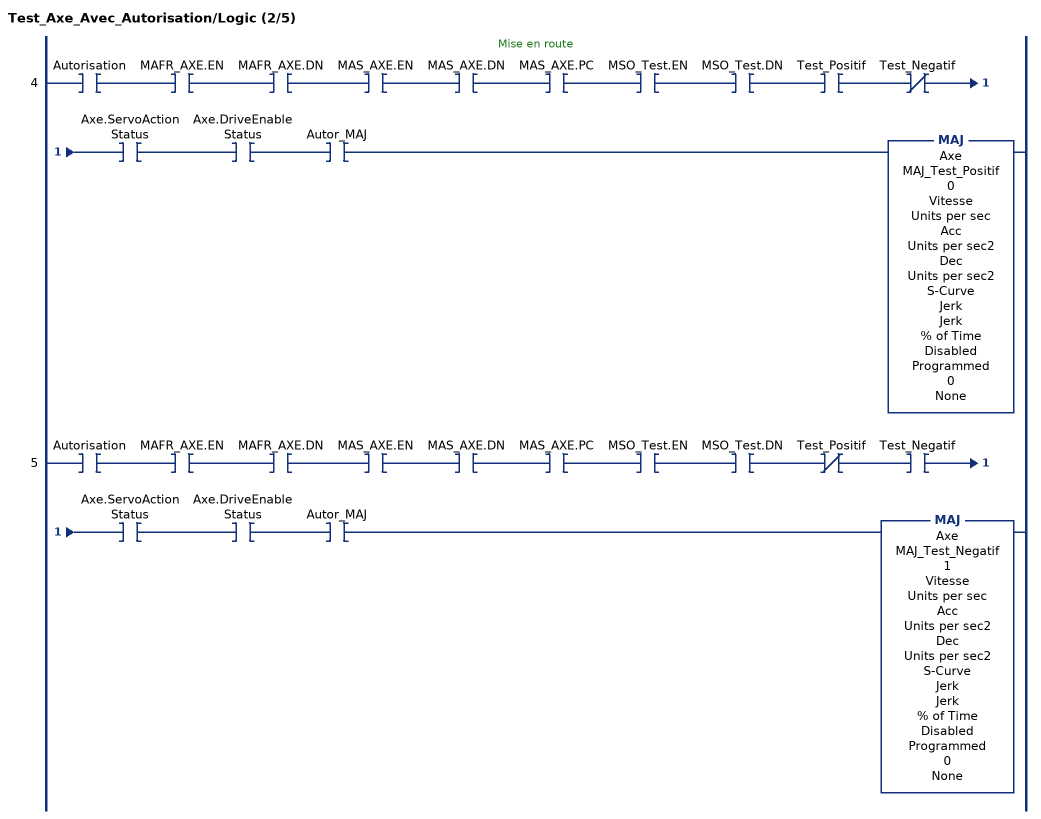
   // Mise en route
   4: XIC(Autorisation)XIC(MAFR_AXE.EN)XIC(MAFR_AXE.DN)XIC(MAS_AXE.EN)XIC(MAS_AXE.DN)XIC(MAS_AXE.PC)XIC(MSO_Test.EN)XIC(MSO_Test.DN)XIC(Test_Positif)XIO(Test_Negatif)XIC(Axe.ServoActionStatus)XIC(Axe.DriveEnableStatus)XIC(Autor_MAJ)MAJ(Axe,MAJ_Test_Positif,0,Vitesse,Units per sec,Acc,Units per sec2,Dec,Units per sec2,S-Curve,Jerk,Jerk,% of Time,Disabled,Programmed,0,None);
   5: XIC(Autorisation)XIC(MAFR_AXE.EN)XIC(MAFR_AXE.DN)XIC(MAS_AXE.EN)XIC(MAS_AXE.DN)XIC(MAS_AXE.PC)XIC(MSO_Test.EN)XIC(MSO_Test.DN)XIO(Test_Positif)XIC(Test_Negatif)XIC(Axe.ServoActionStatus)XIC(Axe.DriveEnableStatus)XIC(Autor_MAJ)MAJ(Axe,MAJ_Test_Negatif,1,Vitesse,Units per sec,Acc,Units per sec2,Dec,Units per sec2,S-Curve,Jerk,Jerk,% of Time,Disabled,Programmed,0,None);
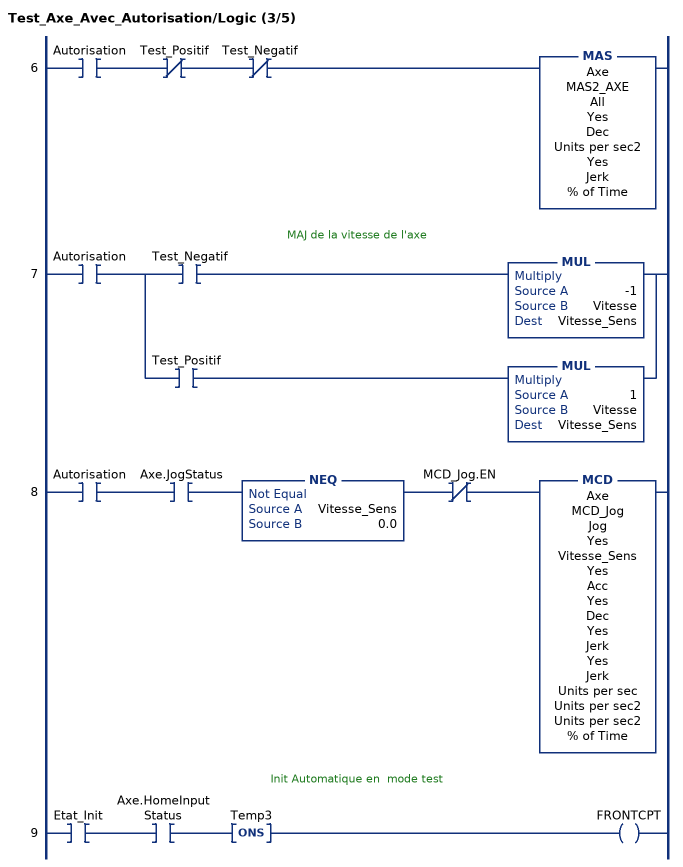
   6: XIC(Autorisation)XIO(Test_Positif)XIO(Test_Negatif)MAS(Axe,MAS2_AXE,All,Yes,Dec,Units per sec2,Yes,Jerk,% of Time);
   // MAJ de la vitesse de l'axe
   7: XIC(Autorisation)[XIC(Test_Negatif) MUL(-1,Vitesse,Vitesse_Sens) ,XIC(Test_Positif) MUL(1,Vitesse,Vitesse_Sens) ];
   8: XIC(Autorisation)XIC(Axe.JogStatus)NEQ(Vitesse_Sens,0.0)XIO(MCD_Jog.EN)MCD(Axe,MCD_Jog,Jog,Yes,Vitesse_Sens,Yes,Acc,Yes,Dec,Yes,Jerk,Yes,Jerk,Units per sec,Units per sec2,Units per sec2,% of Time);
   // Init Automatique en  mode test
   9: XIC(Etat_Init)XIC(Axe.HomeInputStatus)ONS(Temp3)OTE(FRONTCPT);
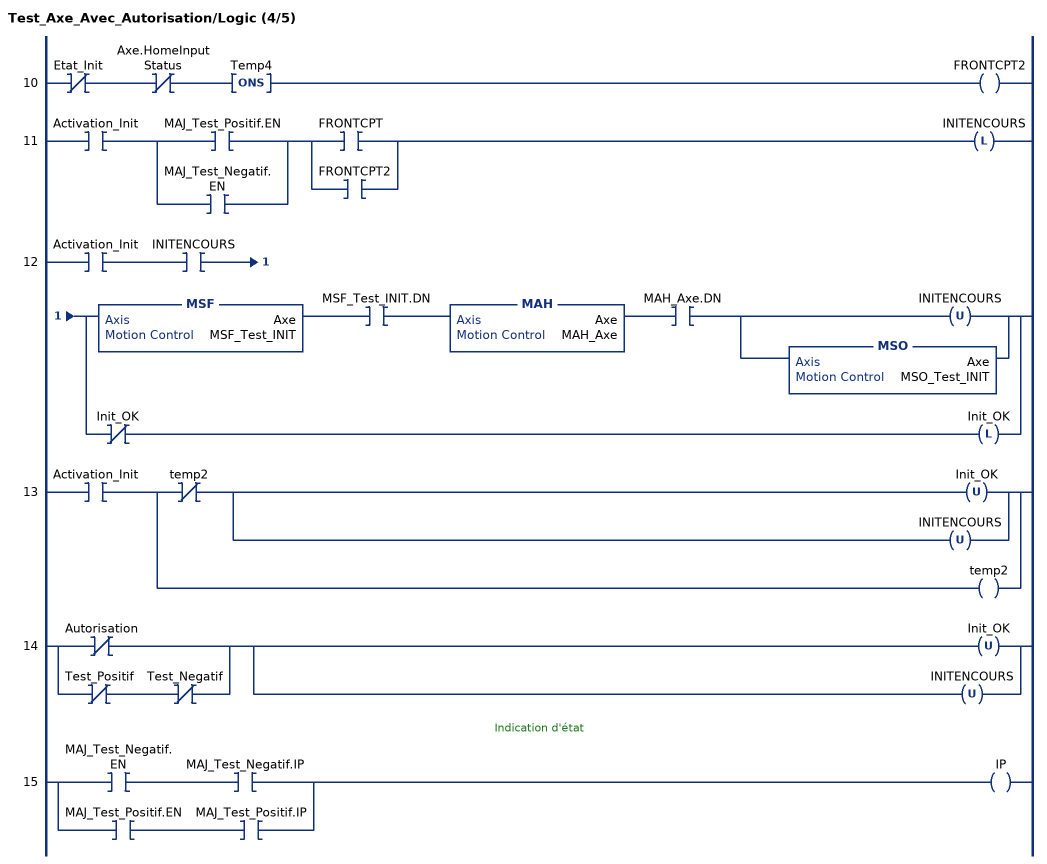
   10: XIO(Etat_Init)XIO(Axe.HomeInputStatus)ONS(Temp4)OTE(FRONTCPT2);
   11: XIC(Activation_Init)[XIC(MAJ_Test_Positif.EN) ,XIC(MAJ_Test_Negatif.EN) ][XIC(FRONTCPT) ,XIC(FRONTCPT2) ]OTL(INITENCOURS);
   12: XIC(Activation_Init)XIC(INITENCOURS)[MSF(Axe,MSF_Test_INIT) XIC(MSF_Test_INIT.DN) MAH(Axe,MAH_Axe) XIC(MAH_Axe.DN) [OTU(INITENCOURS) ,MSO(Axe,MSO_Test_INIT) ] ,XIO(Init_OK) OTL(Init_OK) ];
   13: XIC(Activation_Init)[XIO(temp2) [OTU(Init_OK) ,OTU(INITENCOURS) ] ,OTE(temp2) ];
   14: [XIO(Autorisation) ,XIO(Test_Positif) XIO(Test_Negatif) ][OTU(Init_OK) ,OTU(INITENCOURS) ];
   // Indication d'état
   15: [XIC(MAJ_Test_Negatif.EN) XIC(MAJ_Test_Negatif.IP) ,XIC(MAJ_Test_Positif.EN) XIC(MAJ_Test_Positif.IP) ]OTE(IP);
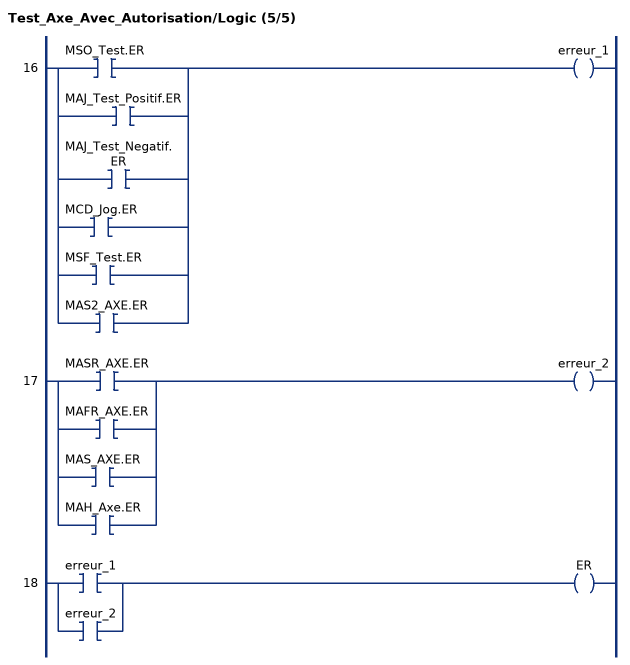
   16: [XIC(MSO_Test.ER) ,[XIC(MAJ_Test_Positif.ER) ,[XIC(MAJ_Test_Negatif.ER) ,[XIC(MCD_Jog.ER) ,[XIC(MSF_Test.ER) ,XIC(MAS2_AXE.ER) ] ] ] ] ]OTE(erreur_1);
   17: [XIC(MASR_AXE.ER) ,[XIC(MAFR_AXE.ER) ,[XIC(MAS_AXE.ER) ,XIC(MAH_Axe.ER) ] ] ]OTE(erreur_2);
   18: [XIC(erreur_1) ,XIC(erreur_2) ]OTE(ER);
END_ROUTINE
END_ADD_ON_INSTRUCTION
